(* IEC 61131-3 sources: CS_4_Aufzugsteuerung/src/Stations/CP112/Steuerung/Class/clsSimpleCounter, 1 file *)

(* ---- clsSimpleCounter.st ---- *)
(*!
<Class
	Name               = "clsSimpleCounter"
	Revision           = "0.0"
	RealtimeTask       = "false"
	CyclicTask         = "true"
	DefCyclictime      = "2 ms"
	BackgroundTask     = "false"
	Sigmatek           = "false"
	OSInterface        = "false"
	HighPriority       = "false"
	Automatic          = "false"
	UpdateMode         = "Prescan"
	SharedCommandTable = "true"
	Objectsize         = "(332,120)">
	<Channels>
		<Server Name="ClassSvr" Visualized="false" Initialize="false" WriteProtected="true" Retentive="false"/>
		<Server Name="Counter" Visualized="false" Initialize="false" WriteProtected="true" Retentive="false"/>
		<Client Name="DigitalIn" Required="true" Internal="false"/>
	</Channels>
</Class>
*)
clsSimpleCounter : CLASS
  //Servers:
	ClassSvr 	: SvrChCmd_DINT;
	Counter 	: SvrCh_DINT;
  //Clients:
	DigitalIn 	: CltCh_DINT;
  //Variables:
		temp 	: DINT;
  //Functions:

	FUNCTION VIRTUAL GLOBAL CyWork
		VAR_INPUT
			EAX 	: UDINT;
		END_VAR
		VAR_OUTPUT
			state (EAX) 	: UDINT;
		END_VAR;
  //Tables:
	FUNCTION @STD
		VAR_OUTPUT
			ret_code	: CONFSTATES;
		END_VAR;
	FUNCTION GLOBAL TAB @CT_;
END_CLASS;

FUNCTION VIRTUAL GLOBAL clsSimpleCounter::CyWork
	VAR_INPUT
		EAX 	: UDINT;
	END_VAR
	VAR_OUTPUT
		state (EAX) 	: UDINT;
	END_VAR

  DigitalIn := DigitalIn.Read();
  Counter := Counter.Read();

  IF temp <> DigitalIn THEN
    temp := DigitalIn;
    Counter += 1;
  END_IF;

  Counter.Write(input:=Counter);

	state := READY;

END_FUNCTION
